LIN {X 0,Y 105.659,Z 342.737,A -85,B 0,C 180,E1 -28297.041,E2 -28297.041} C_VEL
LIN {X 0,Y 105.003,Z 343.905,A -85,B 0,C 180,E1 -28297.746,E2 -28297.746} C_VEL
LIN {X 0,Y 97.324,Z 352.497,A -85,B 0,C 180,E1 -28302.252,E2 -28302.252} C_VEL
LIN {X 0,Y 91.661,Z 358.102,A -85,B 0,C 180,E1 -28306.364,E2 -28306.364} C_VEL
LIN {X 0,Y 85.562,Z 363.557,A -85,B 0,C 180,E1 -28311.971,E2 -28311.971} C_VEL
LIN {X 0,Y 80.28,Z 367.835,A -85,B 0,C 180,E1 -28318.313,E2 -28318.313} C_VEL
LIN {X 0,Y 77.305,Z 370.096,A -85,B 0,C 180,E1 -28322.962,E2 -28322.962} C_VEL
LIN {X 0,Y 74.884,Z 371.926,A -85,B 0,C 180,E1 -28327.949,E2 -28327.949} C_VEL
LIN {X 0,Y 72.17,Z 373.834,A -85,B 0,C 180,E1 -28336.205,E2 -28336.205} C_VEL
LIN {X 0,Y 70.569,Z 374.611,A -85,B 0,C 180,E1 -28340.732,E2 -28340.732} C_VEL
LIN {X 0,Y 66.947,Z 375.27,A -85,B 0,C 180,E1 -28348.413,E2 -28348.413} C_VEL
LIN {X 0,Y 64.706,Z 375.334,A -85,B 0,C 180,E1 -28355.093,E2 -28355.093} C_VEL
LIN {X 0,Y 64.356,Z 375.007,A -85,B 0,C 180,E1 -28360.359,E2 -28360.359} C_VEL
LIN {X 0,Y 64.614,Z 374.789,A -85,B 0,C 180,E1 -28362.098,E2 -28362.098} C_VEL
LIN {X 0,Y 66.21,Z 373.781,A -85,B 0,C 180,E1 -28368.568,E2 -28368.568} C_VEL
LIN {X 0,Y 68.345,Z 372.435,A -85,B 0,C 180,E1 -28374.287,E2 -28374.287} C_VEL
LIN {X 0,Y 72.612,Z 369.585,A -85,B 0,C 180,E1 -28382.163,E2 -28382.163} C_VEL
LIN {X 0,Y 78.012,Z 365.713,A -85,B 0,C 180,E1 -28389.095,E2 -28389.095} C_VEL
LIN {X 0,Y 84.34,Z 360.712,A -85,B 0,C 180,E1 -28395.096,E2 -28395.096} C_VEL
LIN {X 0,Y 91.425,Z 354.402,A -85,B 0,C 180,E1 -28400.238,E2 -28400.238} C_VEL
LIN {X 0,Y 99.645,Z 345.919,A -85,B 0,C 180,E1 -28404.893,E2 -28404.893} C_VEL
LIN {X 0,Y 100.509,Z 344.459,A -85,B 0,C 180,E1 -28405.986,E2 -28405.986} C_VEL
LIN {X 0,Y 101.097,Z 341.851,A -85,B 0,C 180,E1 -28408.693,E2 -28408.693} C_VEL
LIN {X 0,Y 101.373,Z 337.405,A -85,B 0,C 180,E1 -28414.325,E2 -28414.325} C_VEL
LIN {X 0,Y 101.282,Z 333.919,A -85,B 0,C 180,E1 -28419.699,E2 -28419.699} C_VEL
LIN {X 0,Y 101.197,Z 331.666,A -85,B 0,C 180,E1 -28423.871,E2 -28423.871} C_VEL
LIN {X 0,Y 101.125,Z 330.018,A -85,B 0,C 180,E1 -28427.966,E2 -28427.966} C_VEL
LIN {X 0,Y 101.082,Z 328.848,A -85,B 0,C 180,E1 -28432.007,E2 -28432.007} C_VEL
LIN {X 0,Y 101.171,Z 328.163,A -85,B 0,C 180,E1 -28436.016,E2 -28436.016} C_VEL
LIN {X 0,Y 101.358,Z 328.005,A -85,B 0,C 180,E1 -28440,E2 -28440} C_VEL
LIN {X 0,Y 100.921,Z 330.742,A -85,B 0,C 180,E1 -28448.006,E2 -28448.006} C_VEL
LIN {X 0,Y 100.844,Z 334.1,A -85,B 0,C 180,E1 -28454.116,E2 -28454.116} C_VEL
LIN {X 0,Y 100.643,Z 337.262,A -85,B 0,C 180,E1 -28458.315,E2 -28458.315} C_VEL
LIN {X 0,Y 99.996,Z 343.261,A -85,B 0,C 180,E1 -28464.942,E2 -28464.942} C_VEL
LIN {X 0,Y 99.66,Z 345.595,A -85,B 0,C 180,E1 -28467.282,E2 -28467.282} C_VEL
LIN {X 0,Y 98.984,Z 347.565,A -85,B 0,C 180,E1 -28468.862,E2 -28468.862} C_VEL
LIN {X 0,Y 94.615,Z 354.531,A -85,B 0,C 180,E1 -28473.317,E2 -28473.317} C_VEL
LIN {X 0,Y 91.515,Z 358.689,A -85,B 0,C 180,E1 -28476.258,E2 -28476.258} C_VEL
LIN {X 0,Y 84.203,Z 365.626,A -85,B 0,C 180,E1 -28481.307,E2 -28481.307} C_VEL
LIN {X 0,Y 77.66,Z 371.198,A -85,B 0,C 180,E1 -28487.256,E2 -28487.256} C_VEL
LIN {X 0,Y 72.038,Z 375.578,A -85,B 0,C 180,E1 -28494.173,E2 -28494.173} C_VEL
LIN {X 0,Y 68.847,Z 377.901,A -85,B 0,C 180,E1 -28499.31,E2 -28499.31} C_VEL
LIN {X 0,Y 66.337,Z 379.794,A -85,B 0,C 180,E1 -28504.928,E2 -28504.928} C_VEL
LIN {X 0,Y 63.389,Z 382.259,A -85,B 0,C 180,E1 -28517.19,E2 -28517.19} C_VEL
LIN {X 0,Y 62.91,Z 382.899,A -85,B 0,C 180,E1 -28523.587,E2 -28523.587} C_VEL
LIN {X 0,Y 63.058,Z 383.138,A -85,B 0,C 180,E1 -28530.001,E2 -28530.001} C_VEL
LIN {X 0,Y 62.911,Z 382.882,A -85,B 0,C 180,E1 -28536.415,E2 -28536.415} C_VEL
LIN {X 0,Y 63.389,Z 382.231,A -85,B 0,C 180,E1 -28542.812,E2 -28542.812} C_VEL
LIN {X 0,Y 66.337,Z 379.738,A -85,B 0,C 180,E1 -28555.074,E2 -28555.074} C_VEL
LIN {X 0,Y 70.393,Z 376.736,A -85,B 0,C 180,E1 -28563.307,E2 -28563.307} C_VEL
LIN {X 0,Y 75.681,Z 372.695,A -85,B 0,C 180,E1 -28570.546,E2 -28570.546} C_VEL
LIN {X 0,Y 82.592,Z 366.908,A -85,B 0,C 180,E1 -28577.39,E2 -28577.39} C_VEL
LIN {X 0,Y 90.317,Z 359.755,A -85,B 0,C 180,E1 -28582.903,E2 -28582.903} C_VEL
LIN {X 0,Y 92.556,Z 357.135,A -85,B 0,C 180,E1 -28584.715,E2 -28584.715} C_VEL
LIN {X 0,Y 98.277,Z 348.505,A -85,B 0,C 180,E1 -28590.402,E2 -28590.402} C_VEL
LIN {X 0,Y 99.416,Z 346.243,A -85,B 0,C 180,E1 -28591.939,E2 -28591.939} C_VEL
LIN {X 0,Y 100.027,Z 342.168,A -85,B 0,C 180,E1 -28595.98,E2 -28595.98} C_VEL
LIN {X 0,Y 100.546,Z 337.04,A -85,B 0,C 180,E1 -28601.667,E2 -28601.667} C_VEL
LIN {X 0,Y 100.774,Z 332.849,A -85,B 0,C 180,E1 -28607.521,E2 -28607.521} C_VEL
LIN {X 0,Y 100.798,Z 330.508,A -85,B 0,C 180,E1 -28611.984,E2 -28611.984} C_VEL
LIN {X 0,Y 101.283,Z 327.69,A -85,B 0,C 180,E1 -28620,E2 -28620} C_VEL
LIN {X 0,Y 101.028,Z 327.931,A -85,B 0,C 180,E1 -28623.989,E2 -28623.989} C_VEL
LIN {X 0,Y 100.898,Z 328.664,A -85,B 0,C 180,E1 -28628.008,E2 -28628.008} C_VEL
LIN {X 0,Y 100.97,Z 330.149,A -85,B 0,C 180,E1 -28632.971,E2 -28632.971} C_VEL
LIN {X 0,Y 101.111,Z 332.475,A -85,B 0,C 180,E1 -28638.227,E2 -28638.227} C_VEL
LIN {X 0,Y 101.262,Z 336.363,A -85,B 0,C 180,E1 -28644.609,E2 -28644.609} C_VEL
LIN {X 0,Y 101.172,Z 339.737,A -85,B 0,C 180,E1 -28649.096,E2 -28649.096} C_VEL
LIN {X 0,Y 100.711,Z 343.259,A -85,B 0,C 180,E1 -28653.131,E2 -28653.131} C_VEL
LIN {X 0,Y 100.464,Z 344.187,A -85,B 0,C 180,E1 -28654.032,E2 -28654.032} C_VEL
LIN {X 0,Y 99.642,Z 345.663,A -85,B 0,C 180,E1 -28655.165,E2 -28655.165} C_VEL
LIN {X 0,Y 91.464,Z 354.146,A -85,B 0,C 180,E1 -28659.789,E2 -28659.789} C_VEL
LIN {X 0,Y 84.432,Z 360.512,A -85,B 0,C 180,E1 -28664.964,E2 -28664.964} C_VEL
LIN {X 0,Y 78.081,Z 365.559,A -85,B 0,C 180,E1 -28670.944,E2 -28670.944} C_VEL
LIN {X 0,Y 72.63,Z 369.474,A -85,B 0,C 180,E1 -28677.844,E2 -28677.844} C_VEL
LIN {X 0,Y 68.37,Z 372.353,A -85,B 0,C 180,E1 -28685.72,E2 -28685.72} C_VEL
LIN {X 0,Y 65.256,Z 374.301,A -85,B 0,C 180,E1 -28694.971,E2 -28694.971} C_VEL
LIN {X 0,Y 63.73,Z 375.299,A -85,B 0,C 180,E1 -28703.668,E2 -28703.668} C_VEL
LIN {X 0,Y 63.43,Z 375.52,A -85,B 0,C 180,E1 -28709.999,E2 -28709.999} C_VEL
LIN {X 0,Y 64.614,Z 374.789,A -85,B 0,C 180,E1 -28722.098,E2 -28722.098} C_VEL
LIN {X 0,Y 65.225,Z 374.124,A -85,B 0,C 180,E1 -28727.244,E2 -28727.244} C_VEL
LIN {X 0,Y 65.359,Z 372.603,A -85,B 0,C 180,E1 -28735.85,E2 -28735.85} C_VEL
LIN {X 0,Y 66.21,Z 370.87,A -85,B 0,C 180,E1 -28742.598,E2 -28742.598} C_VEL
LIN {X 0,Y 68.082,Z 369.177,A -85,B 0,C 180,E1 -28747.182,E2 -28747.182} C_VEL
LIN {X 0,Y 69.021,Z 368.52,A -85,B 0,C 180,E1 -28748.532,E2 -28748.532} C_VEL
LIN {X 0,Y 74.847,Z 364.583,A -85,B 0,C 180,E1 -28754.768,E2 -28754.768} C_VEL
LIN {X 0,Y 83.199,Z 358.163,A -85,B 0,C 180,E1 -28761.385,E2 -28761.385} C_VEL
LIN {X 0,Y 91.104,Z 351.088,A -85,B 0,C 180,E1 -28766.024,E2 -28766.024} C_VEL
LIN {X 0,Y 94.291,Z 347.893,A -85,B 0,C 180,E1 -28767.664,E2 -28767.664} C_VEL
LIN {X 0,Y 95.153,Z 346.464,A -85,B 0,C 180,E1 -28768.867,E2 -28768.867} C_VEL
LIN {X 0,Y 95.682,Z 344.18,A -85,B 0,C 180,E1 -28771.813,E2 -28771.813} C_VEL
LIN {X 0,Y 96.139,Z 341.108,A -85,B 0,C 180,E1 -28776.292,E2 -28776.292} C_VEL
LIN {X 0,Y 96.363,Z 337.469,A -85,B 0,C 180,E1 -28783.038,E2 -28783.038} C_VEL
LIN {X 0,Y 96.462,Z 335.715,A -85,B 0,C 180,E1 -28787.374,E2 -28787.374} C_VEL
LIN {X 0,Y 96.576,Z 334.531,A -85,B 0,C 180,E1 -28791.631,E2 -28791.631} C_VEL
LIN {X 0,Y 96.745,Z 333.805,A -85,B 0,C 180,E1 -28795.834,E2 -28795.834} C_VEL
LIN {X 0,Y 96.935,Z 333.683,A -85,B 0,C 180,E1 -28800,E2 -28800} C_VEL
LIN {X 0,Y 96.498,Z 334.946,A -85,B 0,C 180,E1 -28804.176,E2 -28804.176} C_VEL
LIN {X 0,Y 96.31,Z 336.529,A -85,B 0,C 180,E1 -28808.392,E2 -28808.392} C_VEL
LIN {X 0,Y 96.024,Z 338.733,A -85,B 0,C 180,E1 -28812.684,E2 -28812.684} C_VEL
LIN {X 0,Y 95.533,Z 341.774,A -85,B 0,C 180,E1 -28817.113,E2 -28817.113} C_VEL
LIN {X 0,Y 94.371,Z 347.49,A -85,B 0,C 180,E1 -28824.065,E2 -28824.065} C_VEL
LIN {X 0,Y 93.811,Z 349.343,A -85,B 0,C 180,E1 -28825.974,E2 -28825.974} C_VEL
LIN {X 0,Y 92.389,Z 351.61,A -85,B 0,C 180,E1 -28827.6,E2 -28827.6} C_VEL
LIN {X 0,Y 87.336,Z 358.245,A -85,B 0,C 180,E1 -28832.335,E2 -28832.335} C_VEL
LIN {X 0,Y 83.54,Z 361.918,A -85,B 0,C 180,E1 -28834.891,E2 -28834.891} C_VEL
LIN {X 0,Y 74.753,Z 369.051,A -85,B 0,C 180,E1 -28841.226,E2 -28841.226} C_VEL
LIN {X 0,Y 68.304,Z 373.823,A -85,B 0,C 180,E1 -28848.026,E2 -28848.026} C_VEL
LIN {X 0,Y 62.83,Z 377.473,A -85,B 0,C 180,E1 -28855.994,E2 -28855.994} C_VEL
LIN {X 0,Y 59.935,Z 379.364,A -85,B 0,C 180,E1 -28862.029,E2 -28862.029} C_VEL
LIN {X 0,Y 56.456,Z 381.83,A -85,B 0,C 180,E1 -28875.584,E2 -28875.584} C_VEL
LIN {X 0,Y 55.836,Z 382.471,A -85,B 0,C 180,E1 -28882.77,E2 -28882.77} C_VEL
LIN {X 0,Y 55.967,Z 382.711,A -85,B 0,C 180,E1 -28890.001,E2 -28890.001} C_VEL
LIN {X 0,Y 55.836,Z 382.453,A -85,B 0,C 180,E1 -28897.232,E2 -28897.232} C_VEL
LIN {X 0,Y 56.457,Z 381.801,A -85,B 0,C 180,E1 -28904.418,E2 -28904.418} C_VEL
LIN {X 0,Y 57.816,Z 380.756,A -85,B 0,C 180,E1 -28911.389,E2 -28911.389} C_VEL
LIN {X 0,Y 59.935,Z 379.306,A -85,B 0,C 180,E1 -28917.973,E2 -28917.973} C_VEL
LIN {X 0,Y 64.537,Z 376.305,A -85,B 0,C 180,E1 -28926.796,E2 -28926.796} C_VEL
LIN {X 0,Y 70.408,Z 372.264,A -85,B 0,C 180,E1 -28934.326,E2 -28934.326} C_VEL
LIN {X 0,Y 78.3,Z 366.165,A -85,B 0,C 180,E1 -28941.55,E2 -28941.55} C_VEL
LIN {X 0,Y 86.158,Z 359.318,A -85,B 0,C 180,E1 -28946.733,E2 -28946.733} C_VEL
LIN {X 0,Y 91.316,Z 352.82,A -85,B 0,C 180,E1 -28951.472,E2 -28951.472} C_VEL
LIN {X 0,Y 93.84,Z 349.09,A -85,B 0,C 180,E1 -28953.993,E2 -28953.993} C_VEL
LIN {X 0,Y 94.707,Z 345.317,A -85,B 0,C 180,E1 -28958.22,E2 -28958.22} C_VEL
LIN {X 0,Y 95.481,Z 341.38,A -85,B 0,C 180,E1 -28963.116,E2 -28963.116} C_VEL
LIN {X 0,Y 95.914,Z 338.533,A -85,B 0,C 180,E1 -28967.302,E2 -28967.302} C_VEL
LIN {X 0,Y 96.217,Z 336.286,A -85,B 0,C 180,E1 -28971.6,E2 -28971.6} C_VEL
LIN {X 0,Y 96.86,Z 333.395,A -85,B 0,C 180,E1 -28980,E2 -28980} C_VEL
LIN {X 0,Y 96.619,Z 333.573,A -85,B 0,C 180,E1 -28984.172,E2 -28984.172} C_VEL
LIN {X 0,Y 96.405,Z 334.348,A -85,B 0,C 180,E1 -28988.384,E2 -28988.384} C_VEL
LIN {X 0,Y 96.314,Z 335.519,A -85,B 0,C 180,E1 -28992.645,E2 -28992.645} C_VEL
LIN {X 0,Y 96.206,Z 337.868,A -85,B 0,C 180,E1 -28998.252,E2 -28998.252} C_VEL
LIN {X 0,Y 96.001,Z 340.913,A -85,B 0,C 180,E1 -29003.744,E2 -29003.744} C_VEL
LIN {X 0,Y 95.437,Z 344.982,A -85,B 0,C 180,E1 -29009.594,E2 -29009.594} C_VEL
LIN {X 0,Y 95.111,Z 346.208,A -85,B 0,C 180,E1 -29011.148,E2 -29011.148} C_VEL
LIN {X 0,Y 94.264,Z 347.658,A -85,B 0,C 180,E1 -29012.402,E2 -29012.402} C_VEL
LIN {X 0,Y 85.821,Z 355.73,A -85,B 0,C 180,E1 -29017.017,E2 -29017.017} C_VEL
LIN {X 0,Y 79.569,Z 360.941,A -85,B 0,C 180,E1 -29021.342,E2 -29021.342} C_VEL
LIN {X 0,Y 72.726,Z 365.986,A -85,B 0,C 180,E1 -29027.431,E2 -29027.431} C_VEL
LIN {X 0,Y 66.736,Z 369.901,A -85,B 0,C 180,E1 -29034.604,E2 -29034.604} C_VEL
LIN {X 0,Y 61.976,Z 372.781,A -85,B 0,C 180,E1 -29043.024,E2 -29043.024} C_VEL
LIN {X 0,Y 59.589,Z 374.15,A -85,B 0,C 180,E1 -29049.277,E2 -29049.277} C_VEL
LIN {X 0,Y 56.88,Z 375.62,A -85,B 0,C 180,E1 -29061.295,E2 -29061.295} C_VEL
LIN {X 0,Y 56.353,Z 375.946,A -85,B 0,C 180,E1 -29069.999,E2 -29069.999} C_VEL
LIN {X 0,Y 57.811,Z 375.164,A -85,B 0,C 180,E1 -29084.071,E2 -29084.071} C_VEL
LIN {X 0,Y 61.957,Z 372.861,A -85,B 0,C 180,E1 -29096.983,E2 -29096.983} C_VEL
LIN {X 0,Y 66.715,Z 370.012,A -85,B 0,C 180,E1 -29105.407,E2 -29105.407} C_VEL
LIN {X 0,Y 69.021,Z 368.52,A -85,B 0,C 180,E1 -29108.532,E2 -29108.532} C_VEL
LIN {X 0,Y 71.648,Z 366.503,A -85,B 0,C 180,E1 -29112.513,E2 -29112.513} C_VEL
LIN {X 0,Y 75.114,Z 362.822,A -85,B 0,C 180,E1 -29119.199,E2 -29119.199} C_VEL
LIN {X 0,Y 79.303,Z 358.555,A -85,B 0,C 180,E1 -29125.054,E2 -29125.054} C_VEL
LIN {X 0,Y 82.829,Z 355.464,A -85,B 0,C 180,E1 -29127.616,E2 -29127.616} C_VEL
LIN {X 0,Y 88.755,Z 350.173,A -85,B 0,C 180,E1 -29130.577,E2 -29130.577} C_VEL
LIN {X 0,Y 89.841,Z 348.674,A -85,B 0,C 180,E1 -29132.007,E2 -29132.007} C_VEL
LIN {X 0,Y 90.785,Z 344.874,A -85,B 0,C 180,E1 -29138.273,E2 -29138.273} C_VEL
LIN {X 0,Y 91.082,Z 343.074,A -85,B 0,C 180,E1 -29142.022,E2 -29142.022} C_VEL
LIN {X 0,Y 91.407,Z 341.23,A -85,B 0,C 180,E1 -29146.664,E2 -29146.664} C_VEL
LIN {X 0,Y 91.71,Z 339.943,A -85,B 0,C 180,E1 -29151.183,E2 -29151.183} C_VEL
LIN {X 0,Y 92.012,Z 339.203,A -85,B 0,C 180,E1 -29155.619,E2 -29155.619} C_VEL
LIN {X 0,Y 92.188,Z 339.13,A -85,B 0,C 180,E1 -29160,E2 -29160} C_VEL
LIN {X 0,Y 91.647,Z 340.461,A -85,B 0,C 180,E1 -29164.509,E2 -29164.509} C_VEL
LIN {X 0,Y 91.259,Z 342.087,A -85,B 0,C 180,E1 -29168.86,E2 -29168.86} C_VEL
LIN {X 0,Y 91.017,Z 343.173,A -85,B 0,C 180,E1 -29171.13,E2 -29171.13} C_VEL
LIN {X 0,Y 90.051,Z 346.617,A -85,B 0,C 180,E1 -29176.619,E2 -29176.619} C_VEL
LIN {X 0,Y 88.832,Z 350.669,A -85,B 0,C 180,E1 -29182.072,E2 -29182.072} C_VEL
LIN {X 0,Y 88.362,Z 351.828,A -85,B 0,C 180,E1 -29183.433,E2 -29183.433} C_VEL
LIN {X 0,Y 87.454,Z 353.175,A -85,B 0,C 180,E1 -29184.526,E2 -29184.526} C_VEL
LIN {X 0,Y 82.349,Z 359.067,A -85,B 0,C 180,E1 -29188.982,E2 -29188.982} C_VEL
LIN {X 0,Y 76.892,Z 363.739,A -85,B 0,C 180,E1 -29192.28,E2 -29192.28} C_VEL
LIN {X 0,Y 69.846,Z 368.905,A -85,B 0,C 180,E1 -29197.137,E2 -29197.137} C_VEL
LIN {X 0,Y 63.176,Z 373.394,A -85,B 0,C 180,E1 -29203.69,E2 -29203.69} C_VEL
LIN {X 0,Y 57.066,Z 377.045,A -85,B 0,C 180,E1 -29211.992,E2 -29211.992} C_VEL
LIN {X 0,Y 53.727,Z 378.934,A -85,B 0,C 180,E1 -29218.451,E2 -29218.451} C_VEL
LIN {X 0,Y 49.572,Z 381.4,A -85,B 0,C 180,E1 -29233.529,E2 -29233.529} C_VEL
LIN {X 0,Y 48.796,Z 382.043,A -85,B 0,C 180,E1 -29241.72,E2 -29241.72} C_VEL
LIN {X 0,Y 48.867,Z 382.283,A -85,B 0,C 180,E1 -29250.001,E2 -29250.001} C_VEL
LIN {X 0,Y 48.796,Z 382.025,A -85,B 0,C 180,E1 -29258.282,E2 -29258.282} C_VEL
LIN {X 0,Y 51.236,Z 380.326,A -85,B 0,C 180,E1 -29274.301,E2 -29274.301} C_VEL
LIN {X 0,Y 53.727,Z 378.875,A -85,B 0,C 180,E1 -29281.551,E2 -29281.551} C_VEL
LIN {X 0,Y 58.971,Z 375.873,A -85,B 0,C 180,E1 -29290.957,E2 -29290.957} C_VEL
LIN {X 0,Y 65.489,Z 371.832,A -85,B 0,C 180,E1 -29298.697,E2 -29298.697} C_VEL
LIN {X 0,Y 74.07,Z 365.733,A -85,B 0,C 180,E1 -29305.881,E2 -29305.881} C_VEL
LIN {X 0,Y 81.053,Z 360.132,A -85,B 0,C 180,E1 -29310.124,E2 -29310.124} C_VEL
LIN {X 0,Y 85.871,Z 354.807,A -85,B 0,C 180,E1 -29314.197,E2 -29314.197} C_VEL
LIN {X 0,Y 88.371,Z 351.583,A -85,B 0,C 180,E1 -29316.569,E2 -29316.569} C_VEL
LIN {X 0,Y 89.65,Z 347.568,A -85,B 0,C 180,E1 -29321.725,E2 -29321.725} C_VEL
LIN {X 0,Y 90.579,Z 344.318,A -85,B 0,C 180,E1 -29326.54,E2 -29326.54} C_VEL
LIN {X 0,Y 91.186,Z 341.859,A -85,B 0,C 180,E1 -29331.133,E2 -29331.133} C_VEL
LIN {X 0,Y 91.604,Z 340.097,A -85,B 0,C 180,E1 -29335.868,E2 -29335.868} C_VEL
LIN {X 0,Y 92.118,Z 338.863,A -85,B 0,C 180,E1 -29340,E2 -29340} C_VEL
LIN {X 0,Y 91.786,Z 339.165,A -85,B 0,C 180,E1 -29345.484,E2 -29345.484} C_VEL
LIN {X 0,Y 91.564,Z 339.766,A -85,B 0,C 180,E1 -29348.831,E2 -29348.831} C_VEL
LIN {X 0,Y 91.275,Z 341.035,A -85,B 0,C 180,E1 -29353.356,E2 -29353.356} C_VEL
LIN {X 0,Y 90.988,Z 342.857,A -85,B 0,C 180,E1 -29357.997,E2 -29357.997} C_VEL
LIN {X 0,Y 90.575,Z 345.259,A -85,B 0,C 180,E1 -29362.828,E2 -29362.828} C_VEL
LIN {X 0,Y 89.77,Z 348.45,A -85,B 0,C 180,E1 -29368.018,E2 -29368.018} C_VEL
LIN {X 0,Y 88.787,Z 349.9,A -85,B 0,C 180,E1 -29369.456,E2 -29369.456} C_VEL
LIN {X 0,Y 80.392,Z 357.263,A -85,B 0,C 180,E1 -29373.847,E2 -29373.847} C_VEL
LIN {X 0,Y 72.532,Z 363.164,A -85,B 0,C 180,E1 -29379.178,E2 -29379.178} C_VEL
LIN {X 0,Y 65.359,Z 367.823,A -85,B 0,C 180,E1 -29385.657,E2 -29385.657} C_VEL
LIN {X 0,Y 59.169,Z 371.378,A -85,B 0,C 180,E1 -29393.565,E2 -29393.565} C_VEL
LIN {X 0,Y 55.743,Z 373.209,A -85,B 0,C 180,E1 -29399.713,E2 -29399.713} C_VEL
LIN {X 0,Y 53.011,Z 374.578,A -85,B 0,C 180,E1 -29406.562,E2 -29406.562} C_VEL
LIN {X 0,Y 50.972,Z 375.552,A -85,B 0,C 180,E1 -29413.992,E2 -29413.992} C_VEL
LIN {X 0,Y 49.285,Z 376.372,A -85,B 0,C 180,E1 -29429.999,E2 -29429.999} C_VEL
LIN {X 0,Y 49.696,Z 376.174,A -85,B 0,C 180,E1 -29438.129,E2 -29438.129} C_VEL
LIN {X 0,Y 50.97,Z 375.591,A -85,B 0,C 180,E1 -29446.007,E2 -29446.007} C_VEL
LIN {X 0,Y 55.725,Z 373.287,A -85,B 0,C 180,E1 -29460.296,E2 -29460.296} C_VEL
LIN {X 0,Y 61.08,Z 370.437,A -85,B 0,C 180,E1 -29469.259,E2 -29469.259} C_VEL
LIN {X 0,Y 67.6,Z 366.565,A -85,B 0,C 180,E1 -29476.697,E2 -29476.697} C_VEL
LIN {X 0,Y 75.005,Z 361.563,A -85,B 0,C 180,E1 -29482.792,E2 -29482.792} C_VEL
LIN {X 0,Y 82.829,Z 355.464,A -85,B 0,C 180,E1 -29487.616,E2 -29487.616} C_VEL
LIN {X 0,Y 84.502,Z 353.806,A -85,B 0,C 180,E1 -29489.093,E2 -29489.093} C_VEL
LIN {X 0,Y 85.474,Z 352.146,A -85,B 0,C 180,E1 -29491.408,E2 -29491.408} C_VEL
LIN {X 0,Y 85.695,Z 351.06,A -85,B 0,C 180,E1 -29493.52,E2 -29493.52} C_VEL
LIN {X 0,Y 85.43,Z 348.252,A -85,B 0,C 180,E1 -29501.18,E2 -29501.18} C_VEL
LIN {X 0,Y 86.253,Z 345.802,A -85,B 0,C 180,E1 -29507.895,E2 -29507.895} C_VEL
LIN {X 0,Y 86.969,Z 344.289,A -85,B 0,C 180,E1 -29515.365,E2 -29515.365} C_VEL
LIN {X 0,Y 87.133,Z 344.295,A -85,B 0,C 180,E1 -29520,E2 -29520} C_VEL
LIN {X 0,Y 86.443,Z 345.618,A -85,B 0,C 180,E1 -29524.663,E2 -29524.663} C_VEL
LIN {X 0,Y 85.709,Z 347.799,A -85,B 0,C 180,E1 -29530.269,E2 -29530.269} C_VEL
LIN {X 0,Y 84.801,Z 350.088,A -85,B 0,C 180,E1 -29534.396,E2 -29534.396} C_VEL
LIN {X 0,Y 83.316,Z 353.604,A -85,B 0,C 180,E1 -29539.719,E2 -29539.719} C_VEL
LIN {X 0,Y 82.798,Z 354.561,A -85,B 0,C 180,E1 -29540.983,E2 -29540.983} C_VEL
LIN {X 0,Y 77.673,Z 359.889,A -85,B 0,C 180,E1 -29545.203,E2 -29545.203} C_VEL
LIN {X 0,Y 69.037,Z 366.361,A -85,B 0,C 180,E1 -29550.083,E2 -29550.083} C_VEL
LIN {X 0,Y 63.947,Z 369.638,A -85,B 0,C 180,E1 -29553.581,E2 -29553.581} C_VEL
LIN {X 0,Y 56.056,Z 374.288,A -85,B 0,C 180,E1 -29561.216,E2 -29561.216} C_VEL
LIN {X 0,Y 51.642,Z 376.617,A -85,B 0,C 180,E1 -29567.122,E2 -29567.122} C_VEL
LIN {X 0,Y 47.785,Z 378.504,A -85,B 0,C 180,E1 -29573.964,E2 -29573.964} C_VEL
LIN {X 0,Y 42.785,Z 380.971,A -85,B 0,C 180,E1 -29590.822,E2 -29590.822} C_VEL
LIN {X 0,Y 41.753,Z 381.614,A -85,B 0,C 180,E1 -29600.311,E2 -29600.311} C_VEL
LIN {X 0,Y 41.761,Z 381.855,A -85,B 0,C 180,E1 -29610.001,E2 -29610.001} C_VEL
LIN {X 0,Y 41.753,Z 381.595,A -85,B 0,C 180,E1 -29619.692,E2 -29619.692} C_VEL
LIN {X 0,Y 42.785,Z 380.941,A -85,B 0,C 180,E1 -29629.181,E2 -29629.181} C_VEL
LIN {X 0,Y 47.784,Z 378.444,A -85,B 0,C 180,E1 -29646.039,E2 -29646.039} C_VEL
LIN {X 0,Y 53.781,Z 375.442,A -85,B 0,C 180,E1 -29655.952,E2 -29655.952} C_VEL
LIN {X 0,Y 62.693,Z 370.325,A -85,B 0,C 180,E1 -29665.292,E2 -29665.292} C_VEL
LIN {X 0,Y 71.878,Z 364.178,A -85,B 0,C 180,E1 -29671.644,E2 -29671.644} C_VEL
LIN {X 0,Y 77.639,Z 359.685,A -85,B 0,C 180,E1 -29674.854,E2 -29674.854} C_VEL
LIN {X 0,Y 82.782,Z 354.336,A -85,B 0,C 180,E1 -29679.049,E2 -29679.049} C_VEL
LIN {X 0,Y 84.051,Z 351.547,A -85,B 0,C 180,E1 -29682.983,E2 -29682.983} C_VEL
LIN {X 0,Y 85.38,Z 348.298,A -85,B 0,C 180,E1 -29688.366,E2 -29688.366} C_VEL
LIN {X 0,Y 85.786,Z 347.18,A -85,B 0,C 180,E1 -29690.57,E2 -29690.57} C_VEL
LIN {X 0,Y 86.366,Z 345.409,A -85,B 0,C 180,E1 -29695.333,E2 -29695.333} C_VEL
LIN {X 0,Y 87.073,Z 344.058,A -85,B 0,C 180,E1 -29700,E2 -29700} C_VEL
LIN {X 0,Y 86.844,Z 344.113,A -85,B 0,C 180,E1 -29704.642,E2 -29704.642} C_VEL
LIN {X 0,Y 86.133,Z 345.535,A -85,B 0,C 180,E1 -29711.72,E2 -29711.72} C_VEL
LIN {X 0,Y 85.887,Z 346.315,A -85,B 0,C 180,E1 -29714.211,E2 -29714.211} C_VEL
LIN {X 0,Y 85.049,Z 349.177,A -85,B 0,C 180,E1 -29721.397,E2 -29721.397} C_VEL
LIN {X 0,Y 84.41,Z 350.849,A -85,B 0,C 180,E1 -29724.602,E2 -29724.602} C_VEL
LIN {X 0,Y 83.627,Z 352.044,A -85,B 0,C 180,E1 -29726.162,E2 -29726.162} C_VEL
LIN {X 0,Y 75.235,Z 358.796,A -85,B 0,C 180,E1 -29730.22,E2 -29730.22} C_VEL
LIN {X 0,Y 68.277,Z 363.592,A -85,B 0,C 180,E1 -29734.564,E2 -29734.564} C_VEL
LIN {X 0,Y 60.489,Z 368.251,A -85,B 0,C 180,E1 -29740.954,E2 -29740.954} C_VEL
LIN {X 0,Y 53.634,Z 371.806,A -85,B 0,C 180,E1 -29749.065,E2 -29749.065} C_VEL
LIN {X 0,Y 49.744,Z 373.637,A -85,B 0,C 180,E1 -29755.587,E2 -29755.587} C_VEL
LIN {X 0,Y 46.604,Z 375.004,A -85,B 0,C 180,E1 -29763.1,E2 -29763.1} C_VEL
LIN {X 0,Y 42.713,Z 376.577,A -85,B 0,C 180,E1 -29780.528,E2 -29780.528} C_VEL
LIN {X 0,Y 42.314,Z 376.731,A -85,B 0,C 180,E1 -29794.758,E2 -29794.758} C_VEL
LIN {X 0,Y 44.206,Z 376.017,A -85,B 0,C 180,E1 -29808.539,E2 -29808.539} C_VEL
LIN {X 0,Y 49.73,Z 373.714,A -85,B 0,C 180,E1 -29824.422,E2 -29824.422} C_VEL
LIN {X 0,Y 55.782,Z 370.863,A -85,B 0,C 180,E1 -29833.863,E2 -29833.863} C_VEL
LIN {X 0,Y 62.944,Z 366.991,A -85,B 0,C 180,E1 -29841.405,E2 -29841.405} C_VEL
LIN {X 0,Y 70.946,Z 361.988,A -85,B 0,C 180,E1 -29847.354,E2 -29847.354} C_VEL
LIN {X 0,Y 79.552,Z 355.672,A -85,B 0,C 180,E1 -29852.06,E2 -29852.06} C_VEL
LIN {X 0,Y 83.638,Z 352.274,A -85,B 0,C 180,E1 -29853.9,E2 -29853.9} C_VEL
LIN {X 0,Y 84.598,Z 350.727,A -85,B 0,C 180,E1 -29856.04,E2 -29856.04} C_VEL
LIN {X 0,Y 85.137,Z 349.462,A -85,B 0,C 180,E1 -29858.408,E2 -29858.408} C_VEL
LIN {X 0,Y 85.43,Z 348.252,A -85,B 0,C 180,E1 -29861.18,E2 -29861.18} C_VEL
LIN {X 0,Y 85.165,Z 347.707,A -85,B 0,C 180,E1 -29863.783,E2 -29863.783} C_VEL
LIN {X 0,Y 84.338,Z 347.775,A -85,B 0,C 180,E1 -29866.409,E2 -29866.409} C_VEL
LIN {X 0,Y 81.638,Z 349.094,A -85,B 0,C 180,E1 -29874.624,E2 -29874.624} C_VEL
LIN {X 0,Y 81.574,Z 349.131,A -85,B 0,C 180,E1 -29875.583,E2 -29875.583} C_VEL
LIN {X 0,Y 81.726,Z 349.174,A -85,B 0,C 180,E1 -29880,E2 -29880} C_VEL
LIN {X 0,Y 80.896,Z 350.555,A -85,B 0,C 180,E1 -29884.984,E2 -29884.984} C_VEL
LIN {X 0,Y 79.949,Z 352.55,A -85,B 0,C 180,E1 -29890.126,E2 -29890.126} C_VEL
LIN {X 0,Y 79.257,Z 353.831,A -85,B 0,C 180,E1 -29892.733,E2 -29892.733} C_VEL
LIN {X 0,Y 77.359,Z 357.011,A -85,B 0,C 180,E1 -29897.943,E2 -29897.943} C_VEL
LIN {X 0,Y 73.366,Z 360.625,A -85,B 0,C 180,E1 -29900.935,E2 -29900.935} C_VEL
LIN {X 0,Y 65.751,Z 365.933,A -85,B 0,C 180,E1 -29904.696,E2 -29904.696} C_VEL
LIN {X 0,Y 57.034,Z 371.083,A -85,B 0,C 180,E1 -29910.394,E2 -29910.394} C_VEL
LIN {X 0,Y 49.088,Z 375.098,A -85,B 0,C 180,E1 -29918.054,E2 -29918.054} C_VEL
LIN {X 0,Y 42.219,Z 378.075,A -85,B 0,C 180,E1 -29928.253,E2 -29928.253} C_VEL
LIN {X 0,Y 36.111,Z 380.541,A -85,B 0,C 180,E1 -29947.094,E2 -29947.094} C_VEL
LIN {X 0,Y 34.753,Z 381.185,A -85,B 0,C 180,E1 -29958.334,E2 -29958.334} C_VEL
LIN {X 0,Y 34.662,Z 381.428,A -85,B 0,C 180,E1 -29970.002,E2 -29970.002} C_VEL
LIN {X 0,Y 34.753,Z 381.166,A -85,B 0,C 180,E1 -29981.669,E2 -29981.669} C_VEL
LIN {X 0,Y 38.656,Z 379.464,A -85,B 0,C 180,E1 -30003.056,E2 -30003.056} C_VEL
LIN {X 0,Y 42.219,Z 378.013,A -85,B 0,C 180,E1 -30011.751,E2 -30011.751} C_VEL
LIN {X 0,Y 49.085,Z 375.011,A -85,B 0,C 180,E1 -30021.954,E2 -30021.954} C_VEL
LIN {X 0,Y 57.051,Z 370.966,A -85,B 0,C 180,E1 -30029.581,E2 -30029.581} C_VEL
LIN {X 0,Y 67.256,Z 364.767,A -85,B 0,C 180,E1 -30036.116,E2 -30036.116} C_VEL
LIN {X 0,Y 73.337,Z 360.437,A -85,B 0,C 180,E1 -30039.127,E2 -30039.127} C_VEL
LIN {X 0,Y 77.312,Z 356.828,A -85,B 0,C 180,E1 -30042.088,E2 -30042.088} C_VEL
LIN {X 0,Y 78.281,Z 355.301,A -85,B 0,C 180,E1 -30044.375,E2 -30044.375} C_VEL
LIN {X 0,Y 79.945,Z 352.314,A -85,B 0,C 180,E1 -30049.874,E2 -30049.874} C_VEL
LIN {X 0,Y 80.817,Z 350.364,A -85,B 0,C 180,E1 -30055.011,E2 -30055.011} C_VEL
LIN {X 0,Y 81.684,Z 348.947,A -85,B 0,C 180,E1 -30060,E2 -30060} C_VEL
LIN {X 0,Y 81.463,Z 348.965,A -85,B 0,C 180,E1 -30064.949,E2 -30064.949} C_VEL
LIN {X 0,Y 80.859,Z 349.834,A -85,B 0,C 180,E1 -30070.011,E2 -30070.011} C_VEL
LIN {X 0,Y 79.7,Z 352.211,A -85,B 0,C 180,E1 -30077.977,E2 -30077.977} C_VEL
LIN {X 0,Y 79.202,Z 353.345,A -85,B 0,C 180,E1 -30080.79,E2 -30080.79} C_VEL
LIN {X 0,Y 78.399,Z 354.376,A -85,B 0,C 180,E1 -30082.533,E2 -30082.533} C_VEL
LIN {X 0,Y 70.392,Z 360.246,A -85,B 0,C 180,E1 -30086.027,E2 -30086.027} C_VEL
LIN {X 0,Y 61.641,Z 365.699,A -85,B 0,C 180,E1 -30091.226,E2 -30091.226} C_VEL
LIN {X 0,Y 53.474,Z 369.974,A -85,B 0,C 180,E1 -30097.946,E2 -30097.946} C_VEL
LIN {X 0,Y 48.51,Z 372.233,A -85,B 0,C 180,E1 -30103.58,E2 -30103.58} C_VEL
LIN {X 0,Y 44.083,Z 374.065,A -85,B 0,C 180,E1 -30110.377,E2 -30110.377} C_VEL
LIN {X 0,Y 40.41,Z 375.432,A -85,B 0,C 180,E1 -30118.548,E2 -30118.548} C_VEL
LIN {X 0,Y 35.754,Z 377.003,A -85,B 0,C 180,E1 -30138.662,E2 -30138.662} C_VEL
LIN {X 0,Y 35.14,Z 377.224,A -85,B 0,C 180,E1 -30149.998,E2 -30149.998} C_VEL
LIN {X 0,Y 35.753,Z 377.026,A -85,B 0,C 180,E1 -30161.335,E2 -30161.335} C_VEL
LIN {X 0,Y 37.548,Z 376.444,A -85,B 0,C 180,E1 -30171.982,E2 -30171.982} C_VEL
LIN {X 0,Y 44.072,Z 374.14,A -85,B 0,C 180,E1 -30189.632,E2 -30189.632} C_VEL
LIN {X 0,Y 50.909,Z 371.289,A -85,B 0,C 180,E1 -30199.4,E2 -30199.4} C_VEL
LIN {X 0,Y 58.782,Z 367.417,A -85,B 0,C 180,E1 -30206.816,E2 -30206.816} C_VEL
LIN {X 0,Y 67.39,Z 362.413,A -85,B 0,C 180,E1 -30212.429,E2 -30212.429} C_VEL
LIN {X 0,Y 76.496,Z 356.096,A -85,B 0,C 180,E1 -30216.742,E2 -30216.742} C_VEL
LIN {X 0,Y 78.49,Z 354.524,A -85,B 0,C 180,E1 -30217.554,E2 -30217.554} C_VEL
LIN {X 0,Y 79.314,Z 353.499,A -85,B 0,C 180,E1 -30219.241,E2 -30219.241} C_VEL
LIN {X 0,Y 80.153,Z 351.504,A -85,B 0,C 180,E1 -30224.749,E2 -30224.749} C_VEL
LIN {X 0,Y 81.006,Z 349.98,A -85,B 0,C 180,E1 -30230.007,E2 -30230.007} C_VEL
LIN {X 0,Y 81.574,Z 349.131,A -85,B 0,C 180,E1 -30235.583,E2 -30235.583} C_VEL
LIN {X 0,Y 80.946,Z 349.723,A -85,B 0,C 180,E1 -30238.244,E2 -30238.244} C_VEL
LIN {X 0,Y 79.554,Z 351.074,A -85,B 0,C 180,E1 -30240.713,E2 -30240.713} C_VEL
LIN {X 0,Y 74.392,Z 356.206,A -85,B 0,C 180,E1 -30248.237,E2 -30248.237} C_VEL
LIN {X 0,Y 74.036,Z 356.655,A -85,B 0,C 180,E1 -30249.214,E2 -30249.214} C_VEL
LIN {X 0,Y 72.405,Z 358.95,A -85,B 0,C 180,E1 -30253.918,E2 -30253.918} C_VEL
LIN {X 0,Y 69.517,Z 361.33,A -85,B 0,C 180,E1 -30256.175,E2 -30256.175} C_VEL
LIN {X 0,Y 59.93,Z 367.34,A -85,B 0,C 180,E1 -30260.257,E2 -30260.257} C_VEL
LIN {X 0,Y 50.793,Z 372.107,A -85,B 0,C 180,E1 -30265.925,E2 -30265.925} C_VEL
LIN {X 0,Y 42.301,Z 375.759,A -85,B 0,C 180,E1 -30273.83,E2 -30273.83} C_VEL
LIN {X 0,Y 37.195,Z 377.645,A -85,B 0,C 180,E1 -30280.907,E2 -30280.907} C_VEL
LIN {X 0,Y 29.667,Z 380.111,A -85,B 0,C 180,E1 -30301.722,E2 -30301.722} C_VEL
LIN {X 0,Y 27.829,Z 380.757,A -85,B 0,C 180,E1 -30315.374,E2 -30315.374} C_VEL
LIN {X 0,Y 27.554,Z 381,A -85,B 0,C 180,E1 -30330.002,E2 -30330.002} C_VEL
LIN {X 0,Y 27.83,Z 380.738,A -85,B 0,C 180,E1 -30344.63,E2 -30344.63} C_VEL
LIN {X 0,Y 32.908,Z 379.034,A -85,B 0,C 180,E1 -30369.847,E2 -30369.847} C_VEL
LIN {X 0,Y 37.195,Z 377.582,A -85,B 0,C 180,E1 -30379.098,E2 -30379.098} C_VEL
LIN {X 0,Y 45.038,Z 374.58,A -85,B 0,C 180,E1 -30389.125,E2 -30389.125} C_VEL
LIN {X 0,Y 53.774,Z 370.533,A -85,B 0,C 180,E1 -30396.19,E2 -30396.19} C_VEL
LIN {X 0,Y 64.69,Z 364.334,A -85,B 0,C 180,E1 -30401.921,E2 -30401.921} C_VEL
LIN {X 0,Y 69.496,Z 361.138,A -85,B 0,C 180,E1 -30403.891,E2 -30403.891} C_VEL
LIN {X 0,Y 72.388,Z 358.738,A -85,B 0,C 180,E1 -30406.144,E2 -30406.144} C_VEL
LIN {X 0,Y 74.396,Z 355.97,A -85,B 0,C 180,E1 -30411.854,E2 -30411.854} C_VEL
LIN {X 0,Y 75.99,Z 353.561,A -85,B 0,C 180,E1 -30420,E2 -30420} C_VEL
LIN {X 0,Y 75.788,Z 353.543,A -85,B 0,C 180,E1 -30425.321,E2 -30425.321} C_VEL
LIN {X 0,Y 74.926,Z 354.516,A -85,B 0,C 180,E1 -30430.813,E2 -30430.813} C_VEL
LIN {X 0,Y 73.751,Z 356.336,A -85,B 0,C 180,E1 -30437.644,E2 -30437.644} C_VEL
LIN {X 0,Y 73.125,Z 356.935,A -85,B 0,C 180,E1 -30438.545,E2 -30438.545} C_VEL
LIN {X 0,Y 64.455,Z 362.656,A -85,B 0,C 180,E1 -30442.052,E2 -30442.052} C_VEL
LIN {X 0,Y 55.271,Z 367.7,A -85,B 0,C 180,E1 -30447.113,E2 -30447.113} C_VEL
LIN {X 0,Y 46.629,Z 371.611,A -85,B 0,C 180,E1 -30454.005,E2 -30454.005} C_VEL
LIN {X 0,Y 38.897,Z 374.492,A -85,B 0,C 180,E1 -30463.718,E2 -30463.718} C_VEL
LIN {X 0,Y 34.553,Z 375.86,A -85,B 0,C 180,E1 -30472.394,E2 -30472.394} C_VEL
LIN {X 0,Y 31.114,Z 376.832,A -85,B 0,C 180,E1 -30483.141,E2 -30483.141} C_VEL
LIN {X 0,Y 28.075,Z 377.649,A -85,B 0,C 180,E1 -30509.998,E2 -30509.998} C_VEL
LIN {X 0,Y 28.837,Z 377.452,A -85,B 0,C 180,E1 -30524.104,E2 -30524.104} C_VEL
LIN {X 0,Y 31.093,Z 376.87,A -85,B 0,C 180,E1 -30536.874,E2 -30536.874} C_VEL
LIN {X 0,Y 38.889,Z 374.565,A -85,B 0,C 180,E1 -30556.292,E2 -30556.292} C_VEL
LIN {X 0,Y 46.604,Z 371.715,A -85,B 0,C 180,E1 -30566.036,E2 -30566.036} C_VEL
LIN {X 0,Y 55.223,Z 367.843,A -85,B 0,C 180,E1 -30572.98,E2 -30572.98} C_VEL
LIN {X 0,Y 64.411,Z 362.839,A -85,B 0,C 180,E1 -30578.039,E2 -30578.039} C_VEL
LIN {X 0,Y 73.087,Z 357.164,A -85,B 0,C 180,E1 -30581.49,E2 -30581.49} C_VEL
LIN {X 0,Y 73.749,Z 356.567,A -85,B 0,C 180,E1 -30582.355,E2 -30582.355} C_VEL
LIN {X 0,Y 75.048,Z 354.654,A -85,B 0,C 180,E1 -30589.205,E2 -30589.205} C_VEL
LIN {X 0,Y 75.922,Z 353.682,A -85,B 0,C 180,E1 -30594.688,E2 -30594.688} C_VEL
LIN {X 0,Y 76.052,Z 353.752,A -85,B 0,C 180,E1 -30600,E2 -30600} C_VEL
LIN {X 0,Y 74.96,Z 355.266,A -85,B 0,C 180,E1 -30605.38,E2 -30605.38} C_VEL
LIN {X 0,Y 74.036,Z 356.655,A -85,B 0,C 180,E1 -30609.214,E2 -30609.214} C_VEL
LIN {X 0,Y 72.815,Z 357.885,A -85,B 0,C 180,E1 -30610.893,E2 -30610.893} C_VEL
LIN {X 0,Y 70.335,Z 359.815,A -85,B 0,C 180,E1 -30612.171,E2 -30612.171} C_VEL
LIN {X 0,Y 67.063,Z 361.936,A -85,B 0,C 180,E1 -30612.832,E2 -30612.832} C_VEL
LIN {X 0,Y 57.863,Z 366.915,A -85,B 0,C 180,E1 -30613.671,E2 -30613.671} C_VEL
LIN {X 0,Y 56.586,Z 367.574,A -85,B 0,C 180,E1 -30614.06,E2 -30614.06} C_VEL
LIN {X 0,Y 48.096,Z 371.677,A -85,B 0,C 180,E1 -30618.232,E2 -30618.232} C_VEL
LIN {X 0,Y 38.784,Z 375.33,A -85,B 0,C 180,E1 -30625.039,E2 -30625.039} C_VEL
LIN {X 0,Y 32.963,Z 377.216,A -85,B 0,C 180,E1 -30631.481,E2 -30631.481} C_VEL
LIN {X 0,Y 23.635,Z 379.683,A -85,B 0,C 180,E1 -30653.511,E2 -30653.511} C_VEL
LIN {X 0,Y 21.018,Z 380.328,A -85,B 0,C 180,E1 -30670.468,E2 -30670.468} C_VEL
LIN {X 0,Y 20.445,Z 380.572,A -85,B 0,C 180,E1 -30690.003,E2 -30690.003} C_VEL
LIN {X 0,Y 21.018,Z 380.309,A -85,B 0,C 180,E1 -30709.538,E2 -30709.538} C_VEL
LIN {X 0,Y 27.814,Z 378.604,A -85,B 0,C 180,E1 -30739.296,E2 -30739.296} C_VEL
LIN {X 0,Y 32.963,Z 377.152,A -85,B 0,C 180,E1 -30748.525,E2 -30748.525} C_VEL
LIN {X 0,Y 41.821,Z 374.149,A -85,B 0,C 180,E1 -30757.564,E2 -30757.564} C_VEL
LIN {X 0,Y 51.3,Z 370.099,A -85,B 0,C 180,E1 -30763.539,E2 -30763.539} C_VEL
LIN {X 0,Y 62.845,Z 363.903,A -85,B 0,C 180,E1 -30768.107,E2 -30768.107} C_VEL
LIN {X 0,Y 67.015,Z 361.227,A -85,B 0,C 180,E1 -30769.688,E2 -30769.688} C_VEL
LIN {X 0,Y 67.918,Z 360.297,A -85,B 0,C 180,E1 -30771.636,E2 -30771.636} C_VEL
LIN {X 0,Y 68.733,Z 359.377,A -85,B 0,C 180,E1 -30774.132,E2 -30774.132} C_VEL
LIN {X 0,Y 70.012,Z 357.878,A -85,B 0,C 180,E1 -30780,E2 -30780} C_VEL
LIN {X 0,Y 69.805,Z 357.837,A -85,B 0,C 180,E1 -30785.779,E2 -30785.779} C_VEL
LIN {X 0,Y 68.641,Z 358.855,A -85,B 0,C 180,E1 -30791.817,E2 -30791.817} C_VEL
LIN {X 0,Y 67.805,Z 359.616,A -85,B 0,C 180,E1 -30794.144,E2 -30794.144} C_VEL
LIN {X 0,Y 58.877,Z 364.877,A -85,B 0,C 180,E1 -30797.262,E2 -30797.262} C_VEL
LIN {X 0,Y 49.247,Z 369.535,A -85,B 0,C 180,E1 -30801.931,E2 -30801.931} C_VEL
LIN {X 0,Y 40.073,Z 373.089,A -85,B 0,C 180,E1 -30808.726,E2 -30808.726} C_VEL
LIN {X 0,Y 34.382,Z 374.919,A -85,B 0,C 180,E1 -30815.146,E2 -30815.146} C_VEL
LIN {X 0,Y 29.264,Z 376.287,A -85,B 0,C 180,E1 -30823.904,E2 -30823.904} C_VEL
LIN {X 0,Y 24.997,Z 377.26,A -85,B 0,C 180,E1 -30835.781,E2 -30835.781} C_VEL
LIN {X 0,Y 21.001,Z 378.075,A -85,B 0,C 180,E1 -30869.997,E2 -30869.997} C_VEL
LIN {X 0,Y 22.037,Z 377.879,A -85,B 0,C 180,E1 -30888.595,E2 -30888.595} C_VEL
LIN {X 0,Y 24.984,Z 377.296,A -85,B 0,C 180,E1 -30904.234,E2 -30904.234} C_VEL
LIN {X 0,Y 34.374,Z 374.991,A -85,B 0,C 180,E1 -30924.864,E2 -30924.864} C_VEL
LIN {X 0,Y 43.048,Z 372.141,A -85,B 0,C 180,E1 -30933.886,E2 -30933.886} C_VEL
LIN {X 0,Y 52.388,Z 368.268,A -85,B 0,C 180,E1 -30939.895,E2 -30939.895} C_VEL
LIN {X 0,Y 62.108,Z 363.265,A -85,B 0,C 180,E1 -30944.12,E2 -30944.12} C_VEL
LIN {X 0,Y 67.833,Z 359.788,A -85,B 0,C 180,E1 -30945.986,E2 -30945.986} C_VEL
LIN {X 0,Y 68.69,Z 359.027,A -85,B 0,C 180,E1 -30948.192,E2 -30948.192} C_VEL
LIN {X 0,Y 69.912,Z 357.972,A -85,B 0,C 180,E1 -30954.23,E2 -30954.23} C_VEL
LIN {X 0,Y 70.067,Z 358.054,A -85,B 0,C 180,E1 -30960,E2 -30960} C_VEL
LIN {X 0,Y 68.73,Z 359.571,A -85,B 0,C 180,E1 -30965.869,E2 -30965.869} C_VEL
LIN {X 0,Y 67.944,Z 360.471,A -85,B 0,C 180,E1 -30968.36,E2 -30968.36} C_VEL
LIN {X 0,Y 67.057,Z 361.395,A -85,B 0,C 180,E1 -30970.333,E2 -30970.333} C_VEL
LIN {X 0,Y 62.843,Z 364.075,A -85,B 0,C 180,E1 -30971.892,E2 -30971.892} C_VEL
LIN {X 0,Y 56.586,Z 367.574,A -85,B 0,C 180,E1 -30974.06,E2 -30974.06} C_VEL
LIN {X 0,Y 51.359,Z 370.047,A -85,B 0,C 180,E1 -30975.454,E2 -30975.454} C_VEL
LIN {X 0,Y 42.061,Z 373.45,A -85,B 0,C 180,E1 -30976.536,E2 -30976.536} C_VEL
LIN {X 0,Y 34.46,Z 375.637,A -85,B 0,C 180,E1 -30977.849,E2 -30977.849} C_VEL
LIN {X 0,Y 28.939,Z 377.023,A -85,B 0,C 180,E1 -30980.846,E2 -30980.846} C_VEL
LIN {X 0,Y 27.215,Z 377.396,A -85,B 0,C 180,E1 -30982.626,E2 -30982.626} C_VEL
LIN {X 0,Y 18.388,Z 379.253,A -85,B 0,C 180,E1 -31000.151,E2 -31000.151} C_VEL
LIN {X 0,Y 14.499,Z 379.9,A -85,B 0,C 180,E1 -31021.011,E2 -31021.011} C_VEL
LIN {X 0,Y 13.331,Z 380.143,A -85,B 0,C 180,E1 -31050.004,E2 -31050.004} C_VEL
LIN {X 0,Y 14.5,Z 379.88,A -85,B 0,C 180,E1 -31078.997,E2 -31078.997} C_VEL
LIN {X 0,Y 23.781,Z 378.174,A -85,B 0,C 180,E1 -31112.454,E2 -31112.454} C_VEL
LIN {X 0,Y 29.864,Z 376.721,A -85,B 0,C 180,E1 -31120.283,E2 -31120.283} C_VEL
LIN {X 0,Y 39.644,Z 373.716,A -85,B 0,C 180,E1 -31127.176,E2 -31127.176} C_VEL
LIN {X 0,Y 49.749,Z 369.668,A -85,B 0,C 180,E1 -31131.459,E2 -31131.459} C_VEL
LIN {X 0,Y 61.942,Z 363.369,A -85,B 0,C 180,E1 -31134.644,E2 -31134.644} C_VEL
LIN {X 0,Y 62.979,Z 362.539,A -85,B 0,C 180,E1 -31136.805,E2 -31136.805} C_VEL
LIN {X 0,Y 63.736,Z 361.837,A -85,B 0,C 180,E1 -31140,E2 -31140} C_VEL
LIN {X 0,Y 63.457,Z 361.796,A -85,B 0,C 180,E1 -31146.359,E2 -31146.359} C_VEL
LIN {X 0,Y 62.528,Z 362.38,A -85,B 0,C 180,E1 -31149.023,E2 -31149.023} C_VEL
LIN {X 0,Y 50.415,Z 368.556,A -85,B 0,C 180,E1 -31152.619,E2 -31152.619} C_VEL
LIN {X 0,Y 40.449,Z 372.466,A -85,B 0,C 180,E1 -31157.127,E2 -31157.127} C_VEL
LIN {X 0,Y 30.854,Z 375.346,A -85,B 0,C 180,E1 -31164.333,E2 -31164.333} C_VEL
LIN {X 0,Y 24.873,Z 376.715,A -85,B 0,C 180,E1 -31172.038,E2 -31172.038} C_VEL
LIN {X 0,Y 19.548,Z 377.687,A -85,B 0,C 180,E1 -31184.02,E2 -31184.02} C_VEL
LIN {X 0,Y 13.913,Z 378.502,A -85,B 0,C 180,E1 -31229.996,E2 -31229.996} C_VEL
LIN {X 0,Y 15.492,Z 378.305,A -85,B 0,C 180,E1 -31256.974,E2 -31256.974} C_VEL
LIN {X 0,Y 19.539,Z 377.722,A -85,B 0,C 180,E1 -31275.998,E2 -31275.998} C_VEL
LIN {X 0,Y 30.84,Z 375.418,A -85,B 0,C 180,E1 -31295.715,E2 -31295.715} C_VEL
LIN {X 0,Y 40.433,Z 372.567,A -85,B 0,C 180,E1 -31302.936,E2 -31302.936} C_VEL
LIN {X 0,Y 50.395,Z 368.693,A -85,B 0,C 180,E1 -31307.472,E2 -31307.472} C_VEL
LIN {X 0,Y 62.601,Z 362.516,A -85,B 0,C 180,E1 -31311.079,E2 -31311.079} C_VEL
LIN {X 0,Y 63.611,Z 361.886,A -85,B 0,C 180,E1 -31313.906,E2 -31313.906} C_VEL
LIN {X 0,Y 63.761,Z 361.999,A -85,B 0,C 180,E1 -31320,E2 -31320} C_VEL
LIN {X 0,Y 63.053,Z 362.64,A -85,B 0,C 180,E1 -31322.875,E2 -31322.875} C_VEL
LIN {X 0,Y 62.036,Z 363.488,A -85,B 0,C 180,E1 -31325.333,E2 -31325.333} C_VEL
LIN {X 0,Y 49.736,Z 369.789,A -85,B 0,C 180,E1 -31328.455,E2 -31328.455} C_VEL
LIN {X 0,Y 39.643,Z 373.809,A -85,B 0,C 180,E1 -31332.831,E2 -31332.831} C_VEL
LIN {X 0,Y 27.215,Z 377.396,A -85,B 0,C 180,E1 -31342.626,E2 -31342.626} C_VEL
LIN {X 0,Y 22.02,Z 378.497,A -85,B 0,C 180,E1 -31348.776,E2 -31348.776} C_VEL
LIN {X 0,Y 16.644,Z 379.215,A -85,B 0,C 180,E1 -31356.032,E2 -31356.032} C_VEL
LIN {X 0,Y 7.246,Z 379.733,A -85,B 0,C 180,E1 -31395.753,E2 -31395.753} C_VEL
LIN {X 0,Y 8.334,Z 379.485,A -85,B 0,C 180,E1 -31457.255,E2 -31457.255} C_VEL
LIN {X 0,Y 14.829,Z 378.79,A -85,B 0,C 180,E1 -31481.427,E2 -31481.427} C_VEL
LIN {X 0,Y 28.267,Z 376.291,A -85,B 0,C 180,E1 -31494.019,E2 -31494.019} C_VEL
LIN {X 0,Y 38.69,Z 373.284,A -85,B 0,C 180,E1 -31497.563,E2 -31497.563} C_VEL
LIN {X 0,Y 51.156,Z 368.343,A -85,B 0,C 180,E1 -31500,E2 -31500} C_VEL
LIN {X 0,Y 56.229,Z 365.894,A -85,B 0,C 180,E1 -31500.664,E2 -31500.664} C_VEL
LIN {X 0,Y 57.384,Z 365.225,A -85,B 0,C 180,E1 -31502.214,E2 -31502.214} C_VEL
LIN {X 0,Y 56.321,Z 365.735,A -85,B 0,C 180,E1 -31503.341,E2 -31503.341} C_VEL
LIN {X 0,Y 45.88,Z 370.39,A -85,B 0,C 180,E1 -31505.303,E2 -31505.303} C_VEL
LIN {X 0,Y 35.511,Z 373.943,A -85,B 0,C 180,E1 -31508.27,E2 -31508.27} C_VEL
LIN {X 0,Y 28.67,Z 375.774,A -85,B 0,C 180,E1 -31511.306,E2 -31511.306} C_VEL
LIN {X 0,Y 21.953,Z 377.142,A -85,B 0,C 180,E1 -31516.168,E2 -31516.168} C_VEL
LIN {X 0,Y 15.483,Z 378.114,A -85,B 0,C 180,E1 -31524.784,E2 -31524.784} C_VEL
LIN {X 0,Y 6.833,Z 378.929,A -85,B 0,C 180,E1 -31589.991,E2 -31589.991} C_VEL
LIN {X 0,Y 9.721,Z 378.732,A -85,B 0,C 180,E1 -31636.289,E2 -31636.289} C_VEL
LIN {X 0,Y 15.476,Z 378.149,A -85,B 0,C 180,E1 -31655.254,E2 -31655.254} C_VEL
LIN {X 0,Y 28.663,Z 375.844,A -85,B 0,C 180,E1 -31668.74,E2 -31668.74} C_VEL
LIN {X 0,Y 38.949,Z 372.992,A -85,B 0,C 180,E1 -31672.939,E2 -31672.939} C_VEL
LIN {X 0,Y 49.346,Z 369.118,A -85,B 0,C 180,E1 -31675.515,E2 -31675.515} C_VEL
LIN {X 0,Y 56.312,Z 365.905,A -85,B 0,C 180,E1 -31676.782,E2 -31676.782} C_VEL
LIN {X 0,Y 57.412,Z 365.384,A -85,B 0,C 180,E1 -31678.08,E2 -31678.08} C_VEL
LIN {X 0,Y 56.228,Z 366.054,A -85,B 0,C 180,E1 -31679.301,E2 -31679.301} C_VEL
LIN {X 0,Y 45.687,Z 370.815,A -85,B 0,C 180,E1 -31680.875,E2 -31680.875} C_VEL
LIN {X 0,Y 35.205,Z 374.472,A -85,B 0,C 180,E1 -31683.492,E2 -31683.492} C_VEL
LIN {X 0,Y 24.423,Z 377.158,A -85,B 0,C 180,E1 -31688.118,E2 -31688.118} C_VEL
LIN {X 0,Y 14.828,Z 378.823,A -85,B 0,C 180,E1 -31698.577,E2 -31698.577} C_VEL
LIN {X 0,Y 8.967,Z 379.471,A -85,B 0,C 180,E1 -31718.404,E2 -31718.404} C_VEL
LIN {X 0,Y 6.238,Z 379.716,A -85,B 0,C 180,E1 -31770.009,E2 -31770.009} C_VEL
LIN {X 0,Y 8.334,Z 379.485,A -85,B 0,C 180,E1 -31817.255,E2 -31817.255} C_VEL
LIN {X 0,Y 9.84,Z 381.484,A -85,B 0,C 180,E1 -31826.296,E2 -31826.296} C_VEL
LIN {X 0,Y 9.84,Z 600,A -85,B 0,C 180,E1 -31826.296,E2 -31826.296} C_VEL
LIN {X 0,Y 9.84,Z 600,A -85,B 0,C 180,E1 -31826.296,E2 -31826.296}

QRS_NEXT_CUT()

QRS_NEXT()
QRS_HOME()

END
